PROGRAM MAIN_Examples
VAR

END_VAR


WareHousingExample();

LabelingExample();

//CamGearExample();

END_PROGRAM

(* stored: Version 1.1.0.1, ProductVersion 3.1.4024.12
   POU MAIN_Examples: Id {171499a4-4ffe-4485-87c4-71eaf38382e6}, SpecialFunc None *)
